KUKA KRL program: e_fraes4.src, e_fraes4.dat

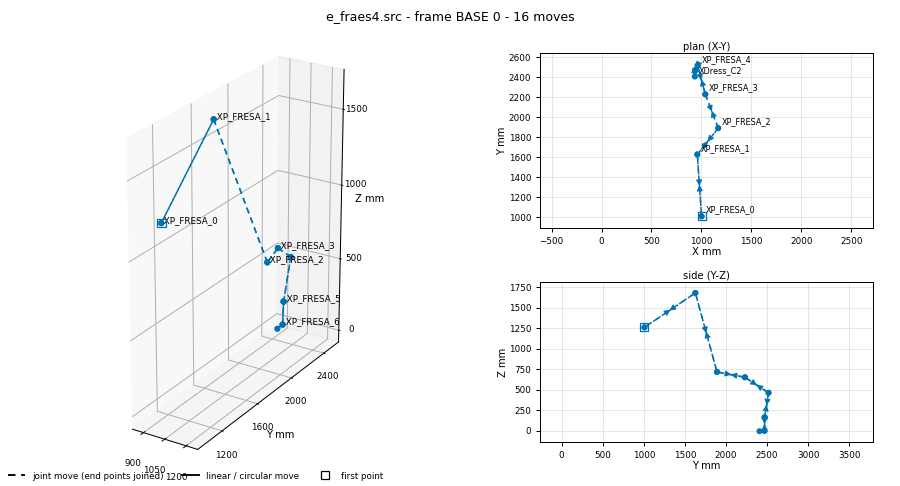
[picture p0: tool path of e_fraes4.src in frame BASE 0, 16 of 18 moves have a stored position in this frame; points joined in program order, loops and branches not executed]
--- e_fraes4.src ---
&ACCESS RVP11
&REL 3
&COMMENT Fresa C2
&PARAM TEMPLATE = C:\KRC\Roboter\Template\vorgabe
&PARAM EDITMASK = *
DEF e_fraes4( )
;FOLD INI;%{PE}%V3.2.0,%MKUKATPBASIS,%CINIT,%VCOMMON,%P
;FOLD BAS INI;%{E}%V3.2.0,%MKUKATPBASIS,%CINIT,%VINIT,%P
GLOBAL INTERRUPT DECL 3 WHEN $STOPMESS==TRUE DO IR_STOPM ( )
INTERRUPT ON 3
BAS (#INITMOV,0 )
;ENDFOLD (BAS INI)
;FOLD A20 INI;%{E}%V3.2.0,%MKUKATPA20,%CINIT,%VINIT,%P
IF ARC20==TRUE THEN
A20 (ARC_INI)
INTERRUPT DECL 6 WHEN $CYCFLAG[3]==FALSE DO A20(TECH_STOP2)
ENDIF
;ENDFOLD (A20 INI)
;FOLD A10 INI;%{E}%V3.2.0,%MKUKATPARC,%CINIT,%VINIT,%P
IF A10_OPTION==#ACTIVE THEN
INTERRUPT DECL 4 WHEN $CYCFLAG[2]==FALSE DO A10 (#APPL_ERROR)
INTERRUPT DECL 7 WHEN A_ARC_SWI==#ACTIVE DO A10 (#ARC_SEAM)
INTERRUPT DECL 5 WHEN A_FLY_ARC==TRUE DO A10 (#HPU_ARC)
INTERRUPT  ON 5
A10_INI ( )
ENDIF
;ENDFOLD (A10 INI)
;FOLD GRIPPER INI;%{E}%V3.2.0,%MKUKATPGRIPPER,%CINIT,%VINIT,%P
USER_GRP(0,DUMMY,DUMMY,GDEFAULT)
;ENDFOLD (GRIPPER INI)
;FOLD SPOT INI;%{E}%V3.2.0,%MKUKATPSPOT,%CINIT,%VINIT,%P
USERSPOT(#INIT)
;ENDFOLD (SPOT INI)
;FOLD TOUCHSENSE INI;%{E}%V3.2.0,%MKUKATPTS,%CINIT,%VINIT,%P
IF H70_OPTION THEN
INTERRUPT DECL 15 WHEN $MEAS_PULSE[TOUCH_I[TOUCH_ACTIVE].IN_NR] DO H70 (6,CD0 )
INTERRUPT DECL 16 WHEN $ZERO_MOVE DO H70 (7,CD0 )
INTERRUPT DECL 17 WHEN $TECHPAR_C[FG_TOUCH,8]>0.5 DO H70 (8,CD0)
H70 (1,CD0 )
ENDIF
;ENDFOLD (TOUCHSENSE INI)
;FOLD USER INI;%{E}%V3.2.0,%MKUKATPUSER,%CINIT,%VINIT,%P
;Make your modifications here
;ENDFOLD (USER INI)
;ENDFOLD (INI)

; Caracterização dos meios de produção:
; Versão Atual:
; 14/09/2015  Name: P13.060-R3 CHANGES: Fresa C2

;FOLD ; PROGRAMA DE QUITACAO DE FRESAGEM DA PINCA C2;%{PE}%R 4.1.16,%MKUKATPBASIS,%CCOMMENT,%VNORMAL,%P 2:PROGRAMA DE QUITACAO DE FRESAGEM DA PINCA C2
;ENDFOLD
chk_w4_wechs_ok ( )        ;VERIFICAÇÃO DE FERRAMENTA: c2

;FOLD PTP P_EXT3  Vel= 100 % DEFAULT;%{PE}%R 4.1.16,%MKUKATPBASIS,%CMOVE,%VPTP,%P 1:PTP, 2:P_EXT3, 3:, 5:100, 7:DEFAULT
$BWDSTART = FALSE
PDAT_ACT=PDEFAULT
BAS(#PTP_DAT)
FDAT_ACT=FP_EXT3
BAS(#FRAMES)
BAS(#VEL_PTP,100)
PTP XP_EXT3
;ENDFOLD

;FOLD PTP P_FRESA_0 CONT Vel= 100 % PDAT9 Tool[4]:Gun C2 Base[0];%{PE}%R 4.1.16,%MKUKATPBASIS,%CMOVE,%VPTP,%P 1:PTP, 2:P_FRESA_0, 3:C_PTP, 5:100, 7:PDAT9
$BWDSTART = FALSE
PDAT_ACT=PPDAT9
BAS(#PTP_DAT)
FDAT_ACT=FP_FRESA_0
BAS(#FRAMES)
BAS(#VEL_PTP,100)
PTP XP_FRESA_0 C_PTP
;ENDFOLD
;FOLD PTP P_FRESA_1 CONT Vel= 100 % PDAT8 Tool[4]:Gun C2 Base[0];%{PE}%R 4.1.16,%MKUKATPBASIS,%CMOVE,%VPTP,%P 1:PTP, 2:P_FRESA_1, 3:C_PTP, 5:100, 7:PDAT8
$BWDSTART = FALSE
PDAT_ACT=PPDAT8
BAS(#PTP_DAT)
FDAT_ACT=FP_FRESA_1
BAS(#FRAMES)
BAS(#VEL_PTP,100)
PTP XP_FRESA_1 C_PTP
;ENDFOLD
;FOLD PTP P_FRESA_2 CONT Vel= 100 % PDAT2 Tool[4]:Gun C2 Base[0];%{PE}%R 4.1.16,%MKUKATPBASIS,%CMOVE,%VPTP,%P 1:PTP, 2:P_FRESA_2, 3:C_PTP, 5:100, 7:PDAT2
$BWDSTART = FALSE
PDAT_ACT=PPDAT2
BAS(#PTP_DAT)
FDAT_ACT=FP_FRESA_2
BAS(#FRAMES)
BAS(#VEL_PTP,100)
PTP XP_FRESA_2 C_PTP
;ENDFOLD
;FOLD PTP P_FRESA_3 CONT Vel= 100 % PDAT7 Tool[4]:Gun C2 Base[0];%{PE}%R 4.1.16,%MKUKATPBASIS,%CMOVE,%VPTP,%P 1:PTP, 2:P_FRESA_3, 3:C_PTP, 5:100, 7:PDAT7
$BWDSTART = FALSE
PDAT_ACT=PPDAT7
BAS(#PTP_DAT)
FDAT_ACT=FP_FRESA_3
BAS(#FRAMES)
BAS(#VEL_PTP,100)
PTP XP_FRESA_3 C_PTP
;ENDFOLD
;FOLD PTP P_FRESA_4 CONT Vel= 100 % PDAT6 Tool[4]:Gun C2 Base[0];%{PE}%R 4.1.16,%MKUKATPBASIS,%CMOVE,%VPTP,%P 1:PTP, 2:P_FRESA_4, 3:C_PTP, 5:100, 7:PDAT6
$BWDSTART = FALSE
PDAT_ACT=PPDAT6
BAS(#PTP_DAT)
FDAT_ACT=FP_FRESA_4
BAS(#FRAMES)
BAS(#VEL_PTP,100)
PTP XP_FRESA_4 C_PTP
;ENDFOLD
;FOLD PTP P_FRESA_5 CONT Vel= 50 % PDAT5 Tool[4]:Gun C2 Base[0];%{PE}%R 4.1.16,%MKUKATPBASIS,%CMOVE,%VPTP,%P 1:PTP, 2:P_FRESA_5, 3:C_PTP, 5:50, 7:PDAT5
$BWDSTART = FALSE
PDAT_ACT=PPDAT5
BAS(#PTP_DAT)
FDAT_ACT=FP_FRESA_5
BAS(#FRAMES)
BAS(#VEL_PTP,50)
PTP XP_FRESA_5 C_PTP
;ENDFOLD
;FOLD LIN P_FRESA_6  Vel= 0.5 m/s CPDAT1 Tool[4]:Gun C2 Base[0];%{PE}%R 4.1.16,%MKUKATPBASIS,%CMOVE,%VLIN,%P 1:LIN, 2:P_FRESA_6, 3:, 5:0.5, 7:CPDAT1
$BWDSTART = FALSE
LDAT_ACT=LCPDAT1
BAS(#CP_DAT)
FDAT_ACT=FP_FRESA_6
BAS(#FRAMES)
BAS(#VEL_CP,0.5)
LIN XP_FRESA_6
;ENDFOLD

;FOLD ; Posicao de fresagem;%{PE}%R 4.1.16,%MKUKATPBASIS,%CCOMMENT,%VNORMAL,%P 2:Posicao de fresagem
;ENDFOLD
;FOLD TIP.LIN_ Dress_C2, Spot Gun 3 , RETR open , Tool[4], Base[0], EXT.TCP=FALSE;%{PE}%MKUKATPUSER
FDAT_ACT=FDress_C2
BAS(#FRAMES)
LIN  XDress_C2
S_ACT.GUN=3
S_ACT.RETR=#opn
S_READY=FALSE
USERSPOT (#DRESS,S_ACT )
WAIT FOR  S_READY
;ENDFOLD

;FOLD LIN P_FRESA_6  Vel= 0.5 m/s CPDAT2 Tool[4]:Gun C2 Base[0];%{PE}%R 4.1.16,%MKUKATPBASIS,%CMOVE,%VLIN,%P 1:LIN, 2:P_FRESA_6, 3:, 5:0.5, 7:CPDAT2
$BWDSTART = FALSE
LDAT_ACT=LCPDAT2
BAS(#CP_DAT)
FDAT_ACT=FP_FRESA_6
BAS(#FRAMES)
BAS(#VEL_CP,0.5)
LIN XP_FRESA_6
;ENDFOLD
;FOLD PTP P_FRESA_5 CONT Vel= 50 % PDAT10 Tool[4]:Gun C2 Base[0];%{PE}%R 4.1.16,%MKUKATPBASIS,%CMOVE,%VPTP,%P 1:PTP, 2:P_FRESA_5, 3:C_PTP, 5:50, 7:PDAT10
$BWDSTART = FALSE
PDAT_ACT=PPDAT10
BAS(#PTP_DAT)
FDAT_ACT=FP_FRESA_5
BAS(#FRAMES)
BAS(#VEL_PTP,50)
PTP XP_FRESA_5 C_PTP
;ENDFOLD

;FOLD ; Test Solda;%{PE}%R 4.1.16,%MKUKATPBASIS,%CCOMMENT,%VNORMAL,%P 2:Test Solda
;ENDFOLD
;FOLD PTP pSoldaC2 PDAT27 SPOT Gun= 3 RETR OPN PgNo1= 253 ACTIVE= 1 Tool[4]:Gun C2 Base[0];%{PE}%R 4.1.12,%MKUKATPSPOT,%CSPOT,%VPTP,%P 1:PTP, 2:pSoldaC2, 3:, 5:100, 7:PDAT27, 10:3, 12:#FIRST, 14:#OPN, 16:253, 18:1, 20:0, 22:0, 24:1, 25:NORMAL1
$BWDSTART = FALSE
PDAT_ACT=PPDAT27
BAS(#PTP_DAT)
FDAT_ACT=FpSoldaC2
BAS(#FRAMES)
BAS(#VEL_PTP,PPDAT27.VEL)
S_ACT.GUN=3
S_ACT.PAIR=SDEFAULT.PAIR
S_ACT.RETR=#OPN
S_ACT.CLO_TM=1
S_ACT.PGNO1=253
S_ACT.PGNO2=SDEFAULT.PGNO2
S_ACT.PRESS1=SDEFAULT.PRESS1
S_ACT.PRESS2=SDEFAULT.PRESS2
S_READY=FALSE
PTP XpSoldaC2
USERSPOT(#SPOT, S_ACT)
WAIT FOR S_READY
;ENDFOLD

;FOLD PTP P_FRESA_4 CONT Vel= 100 % PDAT11 Tool[4]:Gun C2 Base[0];%{PE}%R 4.1.16,%MKUKATPBASIS,%CMOVE,%VPTP,%P 1:PTP, 2:P_FRESA_4, 3:C_PTP, 5:100, 7:PDAT11
$BWDSTART = FALSE
PDAT_ACT=PPDAT11
BAS(#PTP_DAT)
FDAT_ACT=FP_FRESA_4
BAS(#FRAMES)
BAS(#VEL_PTP,100)
PTP XP_FRESA_4 C_PTP
;ENDFOLD
;FOLD PTP P_FRESA_3 CONT Vel= 100 % PDAT12 Tool[4]:Gun C2 Base[0];%{PE}%R 4.1.16,%MKUKATPBASIS,%CMOVE,%VPTP,%P 1:PTP, 2:P_FRESA_3, 3:C_PTP, 5:100, 7:PDAT12
$BWDSTART = FALSE
PDAT_ACT=PPDAT12
BAS(#PTP_DAT)
FDAT_ACT=FP_FRESA_3
BAS(#FRAMES)
BAS(#VEL_PTP,100)
PTP XP_FRESA_3 C_PTP
;ENDFOLD
;FOLD PTP P_FRESA_2 CONT Vel= 100 % PDAT13 Tool[4]:Gun C2 Base[0];%{PE}%R 4.1.16,%MKUKATPBASIS,%CMOVE,%VPTP,%P 1:PTP, 2:P_FRESA_2, 3:C_PTP, 5:100, 7:PDAT13
$BWDSTART = FALSE
PDAT_ACT=PPDAT13
BAS(#PTP_DAT)
FDAT_ACT=FP_FRESA_2
BAS(#FRAMES)
BAS(#VEL_PTP,100)
PTP XP_FRESA_2 C_PTP
;ENDFOLD
;FOLD PTP P_FRESA_1 CONT Vel= 100 % PDAT14 Tool[4]:Gun C2 Base[0];%{PE}%R 4.1.16,%MKUKATPBASIS,%CMOVE,%VPTP,%P 1:PTP, 2:P_FRESA_1, 3:C_PTP, 5:100, 7:PDAT14
$BWDSTART = FALSE
PDAT_ACT=PPDAT14
BAS(#PTP_DAT)
FDAT_ACT=FP_FRESA_1
BAS(#FRAMES)
BAS(#VEL_PTP,100)
PTP XP_FRESA_1 C_PTP
;ENDFOLD
;FOLD PTP P_FRESA_0 CONT Vel= 100 % PDAT15 Tool[4]:Gun C2 Base[0];%{PE}%R 4.1.16,%MKUKATPBASIS,%CMOVE,%VPTP,%P 1:PTP, 2:P_FRESA_0, 3:C_PTP, 5:100, 7:PDAT15
$BWDSTART = FALSE
PDAT_ACT=PPDAT15
BAS(#PTP_DAT)
FDAT_ACT=FP_FRESA_0
BAS(#FRAMES)
BAS(#VEL_PTP,100)
PTP XP_FRESA_0 C_PTP
;ENDFOLD

;FOLD PTP P_EXT3  Vel= 100 % DEFAULT;%{PE}%R 4.1.16,%MKUKATPBASIS,%CMOVE,%VPTP,%P 1:PTP, 2:P_EXT3, 3:, 5:100, 7:DEFAULT
$BWDSTART = FALSE
PDAT_ACT=PDEFAULT
BAS(#PTP_DAT)
FDAT_ACT=FP_EXT3
BAS(#FRAMES)
BAS(#VEL_PTP,100)
PTP XP_EXT3
;ENDFOLD

END

--- e_fraes4.dat ---
&ACCESS RVP11
&REL 3
&COMMENT Fresa C2
&PARAM TEMPLATE = C:\KRC\Roboter\Template\vorgabe
&PARAM EDITMASK = *
DEFDAT  E_FRAES4
;FOLD EXTERNAL DECLARATIONS;%{PE}%V3.2.0,%MKUKATPBASIS,%CEXT,%VCOMMON,%P
;FOLD BAS EXT;%{PE}%V3.2.0,%MKUKATPBASIS,%CEXT,%VEXT,%P
EXT  BAS (BAS_COMMAND  :IN,REAL  :IN )
DECL INT SUCCESS
;ENDFOLD
;FOLD A10 EXT;%{E}%V3.2.0,%MKUKATPARC,%CEXT,%VEXT,%P
EXT  A10 (A_CMD_T  :IN,A_STRT_T  :IN,A_WELD_T  :IN,A_END_T  :IN,INT  :IN )
;ENDFOLD
;FOLD A20 EXT;%{E}%V3.2.0,%MKUKATPA20,%CEXT,%VEXT,%P
EXT  A20 (INT  :IN,WELD_ST  :IN,WELD_FI  :IN,INT  :IN )
;ENDFOLD
;FOLD GRIPPER EXT;%{E}%V3.2.0,%MKUKATPGRIPPER,%CEXT,%VEXT,%P
EXT  H50 (INT  :IN,INT  :IN,INT  :IN,GRP_TYP  :IN )
;ENDFOLD
;FOLD SPOT EXT;%{E}%V3.2.0,%MKUKATPSPOT,%CEXT,%VEXT,%P
EXT  USERSPOT (S_COMMAND  :IN,SPOT_TYPE  :IN )
;ENDFOLD
;FOLD TOUCHSENSE EXT;%{E}%V3.2.0,%MKUKATPTS,%CEXT,%VEXT,%P
EXT  H70 (INT  :IN,SRCH_TYP_2  :OUT,E6POS  :IN,SRCH_TYP_3  :IN,SRCH_TYP_2  :IN,SRCH_TYP_2  :IN,SRCH_TYP_2  :IN,SRCH_TYP_2  :IN,SRCH_TYP_2  :IN,INT  :IN )
;ENDFOLD
;FOLD USER EXT;%{E}%V3.2.0,%MKUKATPUSER,%CEXT,%VEXT,%P
;Make here your modifications
;ENDFOLD
;ENDFOLD

DECL FDAT FDress_C1={TOOL_NO 1,BASE_NO 0,IPO_FRAME #BASE}
DECL E6POS XDress_C1={x 881.376221,y 2683.7771,z 38.1912918,a -179.760803,b -37.8648911,c -89.5162582,s 2,t 11,e1 0.0,e2 0.0,e3 0.0,e4 0.0,e5 0.0,e6 0.0}
DECL BASIS_SUGG_T LAST_BASIS={POINT1[] "P_FRESA_0               ",POINT2[] "P_FRESA_0               ",CP_PARAMS[] "CPDAT0                  ",PTP_PARAMS[] "PDAT15                  ",CONT[] "C_PTP                   ",CP_VEL[] "2.0                     ",PTP_VEL[] "100                     "}
DECL E6POS XP1={x 827.614929,y 1421.08606,z 1395.94604,a 170.888901,b 15.6599102,c -34.8352013,s 2,t 3,e1 0.0,e2 0.0,e3 0.0,e4 0.0,e5 0.0,e6 0.0}
DECL FDAT FP1={TOOL_NO 4,BASE_NO 0,IPO_FRAME #BASE}
DECL PDAT PPDAT1={VEL 100.0,ACC 85.0,APO_DIST 100.0}
DECL E6POS XP2={x 1168.39001,y 1890.02698,z 716.494629,a -95.8133774,b 32.5636597,c -4.32911777,s 2,t 11,e1 0.0,e2 0.0,e3 0.0,e4 0.0,e5 0.0,e6 0.0}
DECL FDAT FP2={TOOL_NO 4,BASE_NO 0,IPO_FRAME #BASE}
DECL PDAT PPDAT2={VEL 100.0,ACC 85.0,APO_DIST 100.0}
DECL FDAT FDress_C2={TOOL_NO 4,BASE_NO 0,IPO_FRAME #BASE}
DECL E6POS XDress_C2={x 933.528687,y 2406.60791,z -4.19509077,a -175.626495,b 82.3356628,c -87.1386871,s 2,t 11,e1 0.0,e2 0.0,e3 0.0,e4 0.0,e5 0.0,e6 0.0}
DECL E6POS XP3={x 935.705872,y 2467.4729,z 0.707535207,a -176.571594,b 82.3351364,c -87.0820236,s 2,t 11,e1 0.0,e2 0.0,e3 0.0,e4 0.0,e5 0.0,e6 0.0}
DECL FDAT FP3={TOOL_NO 4,BASE_NO 0,IPO_FRAME #BASE}
DECL PDAT PPDAT3={VEL 100.0,ACC 85.0,APO_DIST 10.0}
DECL LDAT LCPDAT1={VEL 2.0,ACC 95.0,APO_DIST 100.0,APO_FAC 50.0}
DECL E6POS XP4={x 935.705872,y 2467.4729,z 0.707535207,a -176.571594,b 82.3351364,c -87.0820236,s 2,t 11,e1 0.0,e2 0.0,e3 0.0,e4 0.0,e5 0.0,e6 0.0}
DECL FDAT FP4={TOOL_NO 4,BASE_NO 0,IPO_FRAME #BASE}
DECL PDAT PPDAT4={VEL 100.0,ACC 85.0,APO_DIST 10.0}
DECL LDAT LCPDAT2={VEL 2.0,ACC 95.0,APO_DIST 100.0,APO_FAC 50.0}
DECL E6POS XP5={x 943.22113,y 2472.06006,z 162.966599,a -158.9039,b 82.209877,c -71.30616,s 2,t 11,e1 0.0,e2 0.0,e3 0.0,e4 0.0,e5 0.0,e6 0.0}
DECL FDAT FP5={TOOL_NO 4,BASE_NO 0,IPO_FRAME #BASE}
DECL PDAT PPDAT5={VEL 100.0,ACC 85.0,APO_DIST 10.0}
DECL E6POS XP6={x 1056.73499,y 2435.58398,z 462.902588,a -104.188698,b 65.2757034,c -16.0155602,s 2,t 11,e1 0.0,e2 0.0,e3 0.0,e4 0.0,e5 0.0,e6 0.0}
DECL FDAT FP6={TOOL_NO 4,BASE_NO 0,IPO_FRAME #BASE}
DECL PDAT PPDAT6={VEL 100.0,ACC 85.0,APO_DIST 10.0}
DECL E6POS XP7={x 1102.30103,y 2072.82202,z 676.347778,a -92.1818008,b 39.0851707,c -7.44022894,s 2,t 11,e1 0.0,e2 0.0,e3 0.0,e4 0.0,e5 0.0,e6 0.0}
DECL FDAT FP7={TOOL_NO 4,BASE_NO 0,IPO_FRAME #BASE}
DECL PDAT PPDAT7={VEL 100.0,ACC 85.0,APO_DIST 10.0}
DECL E6POS XP8={x 988.333923,y 1696.00403,z 1769.31396,a 162.901505,b 22.7600594,c -58.7482109,s 2,t 3,e1 0.0,e2 0.0,e3 0.0,e4 0.0,e5 0.0,e6 0.0}
DECL FDAT FP8={TOOL_NO 4,BASE_NO 0,IPO_FRAME #BASE}
DECL PDAT PPDAT8={VEL 100.0,ACC 85.0,APO_DIST 10.0}
DECL E6POS XP_FRESA_1={x 958.960571,y 1626.84399,z 1677.80701,a 163.379105,b 20.4552402,c -57.0116806,s 2,t 11,e1 0.0,e2 0.0,e3 0.0,e4 0.0,e5 0.0,e6 0.0}
DECL FDAT FP_FRESA_1={TOOL_NO 4,BASE_NO 0,IPO_FRAME #BASE}
DECL E6POS XP_FRESA_0={x 1001.58002,y 1007.427,z 1259.08997,a 45.3985405,b -24.9993,c -0.0984198973,s 2,t 35,e1 0.0,e2 0.0,e3 0.0,e4 0.0,e5 0.0,e6 0.0}
DECL FDAT FP_FRESA_0={TOOL_NO 4,BASE_NO 0,IPO_FRAME #BASE}
DECL PDAT PPDAT9={VEL 100.0,ACC 85.0,APO_DIST 10.0}
DECL E6POS XP_FRESA_2={x 1168.39294,y 1890.02295,z 716.540405,a -95.8144531,b 32.5642509,c -4.32911396,s 2,t 11,e1 0.0,e2 0.0,e3 0.0,e4 0.0,e5 0.0,e6 0.0}
DECL FDAT FP_FRESA_2={TOOL_NO 4,BASE_NO 0,IPO_FRAME #BASE}
DECL E6POS XP_FRESA_3={x 1039.17505,y 2229.25708,z 651.841309,a -91.2074966,b 48.0764389,c -9.61500168,s 2,t 11,e1 0.0,e2 0.0,e3 0.0,e4 0.0,e5 0.0,e6 0.0}
DECL FDAT FP_FRESA_3={TOOL_NO 4,BASE_NO 0,IPO_FRAME #BASE}
DECL E6POS XP_FRESA_4={x 961.768372,y 2517.12305,z 463.016693,a -99.9168777,b 61.3115616,c -24.4062309,s 2,t 11,e1 0.0,e2 0.0,e3 0.0,e4 0.0,e5 0.0,e6 0.0}
DECL FDAT FP_FRESA_4={TOOL_NO 4,BASE_NO 0,IPO_FRAME #BASE}
DECL E6POS XP_FRESA_5={x 940.301514,y 2469.88501,z 163.929993,a -148.145203,b 81.1281891,c -61.1321487,s 2,t 11,e1 0.0,e2 0.0,e3 0.0,e4 0.0,e5 0.0,e6 0.0}
DECL FDAT FP_FRESA_5={TOOL_NO 4,BASE_NO 0,IPO_FRAME #BASE}
DECL E6POS XP_FRESA_6={x 935.760803,y 2467.54102,z 0.828034401,a -173.064301,b 85.1552277,c -83.9172363,s 2,t 11,e1 0.0,e2 0.0,e3 0.0,e4 0.0,e5 0.0,e6 0.0}
DECL FDAT FP_FRESA_6={TOOL_NO 4,BASE_NO 0,IPO_FRAME #BASE}
DECL E6POS XP_FRESA_7={x 943.22113,y 2472.06006,z 162.966599,a -158.9039,b 82.209877,c -71.30616,s 2,t 11,e1 0.0,e2 0.0,e3 0.0,e4 0.0,e5 0.0,e6 0.0}
DECL FDAT FP_FRESA_7={TOOL_NO 4,BASE_NO 0,IPO_FRAME #BASE}
DECL PDAT PPDAT10={VEL 100.0,ACC 85.0,APO_DIST 10.0}
DECL E6POS XP_FRESA_8={x 1056.64404,y 2435.61108,z 463.251007,a -104.184502,b 65.2779236,c -16.0228004,s 2,t 11,e1 0.0,e2 0.0,e3 0.0,e4 0.0,e5 0.0,e6 0.0}
DECL FDAT FP_FRESA_8={TOOL_NO 4,BASE_NO 0,IPO_FRAME #BASE}
DECL PDAT PPDAT11={VEL 100.0,ACC 85.0,APO_DIST 10.0}
DECL PDAT PPDAT12={VEL 100.0,ACC 85.0,APO_DIST 10.0}
DECL PDAT PPDAT13={VEL 100.0,ACC 85.0,APO_DIST 10.0}
DECL PDAT PPDAT14={VEL 100.0,ACC 85.0,APO_DIST 10.0}
DECL PDAT PPDAT15={VEL 100.0,ACC 85.0,APO_DIST 10.0}
DECL E6POS XpSoldaX3={x 919.960388,y 2394.21899,z 117.4888,a -15.7696199,b 86.138443,c -102.699402,s 6,t 51,e1 0.0,e2 0.0,e3 0.0,e4 0.0,e5 0.0,e6 0.0}
DECL FDAT FpSoldaX3={TOOL_NO 2,BASE_NO 0,IPO_FRAME #BASE}
DECL PDAT PPDAT27={VEL 50.0,ACC 100.0,APO_DIST 100.0}
DECL SPOT_TYPE SNORMAL1
DECL SPOT_SUGG_T LAST_SPOT={GUN[] " 1                      ",RETR_CMD[] "#OPN                    ",CHOISE[] "#FIRST                  ",CLO_TM[] "1                       ",PGNO1[] " 1                      ",PRESS1[] "0                       ",PGNO2[] " 1                      ",PRESS2[] "0                       ",SPOT_PARAMS[] "NORMAL                  "}
DECL E6POS XpSoldaC2={x 940.335815,y 2469.854,z 163.897903,a -148.145203,b 81.1270294,c -61.1313705,s 2,t 11,e1 0.0,e2 0.0,e3 0.0,e4 0.0,e5 0.0,e6 0.0}
DECL FDAT FpSoldaC2={TOOL_NO 4,BASE_NO 0,IPO_FRAME #BASE}
ENDDAT
